FUNCTION_BLOCK DoppelLauflicht
VAR_INPUT
END_VAR
VAR_OUTPUT
END_VAR
VAR
	Blinker: TON;
	Zaehler : WORD;
END_VAR


Blinker(IN:= NOT Blinker.Q, PT:= T#100MS );

IF Blinker.Q THEN	Zaehler := Zaehler + 1;END_IF
IF Zaehler > 7 THEN Zaehler := 0;END_IF

dSub.DQB_1_8 := SHL(1, Zaehler);
dSub.DQB_9_16 := SHL(1, 7 - Zaehler);

END_FUNCTION_BLOCK

(* stored: Version 1.1.0.1, ProductVersion 3.1.4022.7
   POU DoppelLauflicht: Id {97617c5f-98a6-4cfd-b852-d438d6d3173c}, SpecialFunc None *)
